// TwinCAT 3 PLC project StructPassDemo
// ProgramVersion: 3.1.4023.0
// libraries:
//   Tc2_Standard, * (Beckhoff Automation GmbH)
//   Tc2_System, * (Beckhoff Automation GmbH)
//   Tc3_Module, * (Beckhoff Automation GmbH)
// project tree:
//   DUTs/ MotorOutputVariables.TcDUT, MotorInputVariables.TcDUT
//   / PlcTask.TcTTO
//   POUs/ MAIN.TcPOU, Motor.TcPOU, Plc_Prog.TcPOU
// real-time tasks:
//   TASK PlcTask: cycle T#10ms, priority 20, ADS port 350

CONFIGURATION StructPassDemo
    RESOURCE PLC ON TwinCAT3
        TASK PlcTask(INTERVAL := T#10ms, PRIORITY := 20);
        PROGRAM MAIN WITH PlcTask : MAIN;
    END_RESOURCE
END_CONFIGURATION

// ---- DUTs/MotorOutputVariables.TcDUT
TYPE MotorOutputVariables :
STRUCT
	Coil : BOOL;
END_STRUCT
END_TYPE

// ---- DUTs/MotorInputVariables.TcDUT
TYPE MotorInputVariables :
STRUCT
	Start : BOOL;
	Stop : BOOL;
	Oveload : BOOL;
	
END_STRUCT
END_TYPE

// ---- POUs/MAIN.TcPOU
PROGRAM MAIN
VAR
END_VAR

Plc_Prog();

END_PROGRAM

// ---- POUs/Plc_Prog.TcPOU
PROGRAM Plc_Prog
VAR
	Motor1 : Motor;
	Motor2 : Motor;
	Motor3 : Motor;
	
	Motor1InputVariables : MotorInputVariables;
	Motor2InputVariables : MotorInputVariables;
	Motor3InputVariables : MotorInputVariables;
	
	Motor1OutputVariables : MotorOutputVariables;
	Motor2OutputVariables : MotorOutputVariables;
	Motor3OutputVariables : MotorOutputVariables;
END_VAR

Motor1(MotorInputs:=Motor1InputVariables, MotorOutputs=>Motor1OutputVariables);
Motor1(MotorInputs:=Motor2InputVariables, MotorOutputs=>Motor2OutputVariables);
Motor1(MotorInputs:=Motor3InputVariables, MotorOutputs=>Motor3OutputVariables);

END_PROGRAM

// ---- POUs/Motor.TcPOU
FUNCTION_BLOCK Motor
VAR_INPUT
	MotorInputs : MotorInputvariables;
END_VAR
VAR_OUTPUT
	MotorOutputs : MotorOutputVariables;
END_VAR
VAR
	Start : BOOL;
	Stop : BOOL;
	
END_VAR

Start := MotorInputs.Start;
Stop := MotorInputs.Stop;

IF Start AND Stop = FALSE AND MotorInputs.Oveload = FALSE THEN
	MotorOutputs.Coil := TRUE;
ELSE
	MotorOutputs.Coil := FALSE;
	
END_IF

END_FUNCTION_BLOCK
